PROGRAM MAIN
VAR

END_VAR


P_TextModeRead();

P_TextModeWrite();

END_PROGRAM

(* stored: Version 1.1.0.1, ProductVersion 3.1.4022.9
   POU MAIN: Id {57f19cc2-6624-4d85-bf79-2cb18e725034}, SpecialFunc None *)
